% RSLogix 500 project SOL7.RSS, saved by version 8.30.00.16 %
PROJECT "PROJ7"    % processor: Bul.1763 MicroLogix 1100 Series B %

PROGRAM FILES
  LAD 2 "MAIN"  6 rungs
  LAD 3 "IO"  5 rungs
  LAD 4 "CONTROL"  3 rungs
  LAD 5 "CALIBRATE"  8 rungs
  LAD 6 "CYCLE"  2 rungs

DATA FILES
  O0 OUTPUT  4 elements
  I1 INPUT  6 elements
  S2 STATUS  66 elements
  B3 BINARY  1 elements
  T4 TIMER  4 elements
  C5 COUNTER  2 elements
  R6 CONTROL  1 elements
  N7 INTEGER  8 elements
  F8 FLOAT  9 elements

LADDER 2 "MAIN"
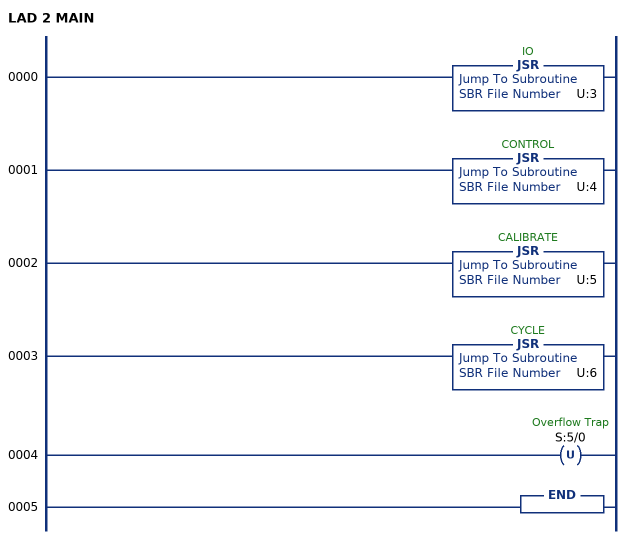
% Rung: 0 %
SOR JSR U:3 EOR
%   U:3  "IO" %
% Rung: 1 %
SOR JSR U:4 EOR
%   U:4  "CONTROL" %
% Rung: 2 %
SOR JSR U:5 EOR
%   U:5  "CALIBRATE" %
% Rung: 3 %
SOR JSR U:6 EOR
%   U:6  "CYCLE" %
% Rung: 4 %
SOR OTU S:5/0 EOR
%   S:5/0  "Overflow Trap" %
% Rung: 5 %
SOR END EOR

LADDER 3 "IO"
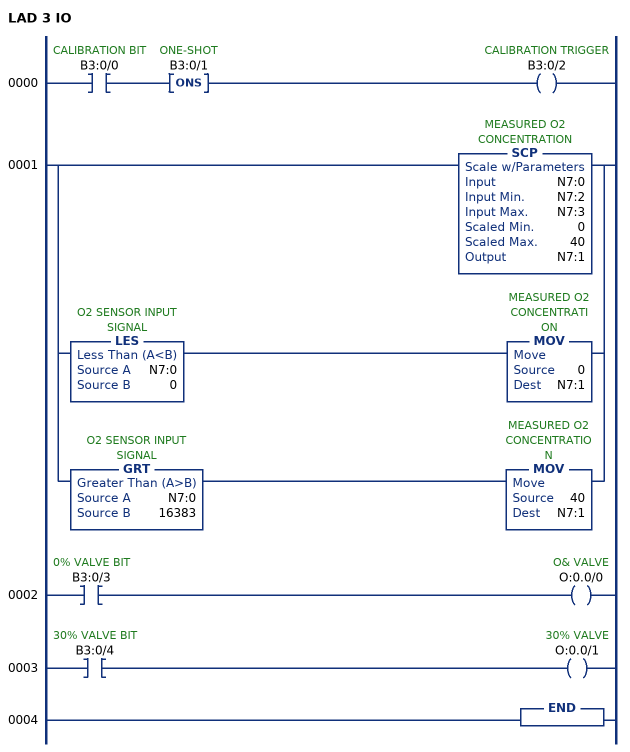
% Rung: 0 %
SOR XIC B3:0/0 ONS B3:0/1 OTE B3:0/2 EOR
%   B3:0/0  "CALIBRATION BIT" %
%   B3:0/1  "ONE-SHOT" %
%   B3:0/2  "CALIBRATION TRIGGER" %
% Rung: 1 %
SOR BST SCP N7:0 N7:2 N7:3 0 40 N7:1 NXB LES N7:0 0 MOV 0 N7:1 NXB GRT N7:0 16383 MOV 40 N7:1 BND EOR
%   N7:0  "O2 SENSOR INPUT SIGNAL" %
%   N7:2  "O2 INPUT MIN" %
%   N7:3  "O2 INPUT MAX" %
%   N7:1  "MEASURED O2 CONCENTRATION" %
% Rung: 2 %
SOR XIC B3:0/3 OTE O:0.0/0 EOR
%   B3:0/3  "0% VALVE BIT" %
%   O:0.0/0  "O& VALVE" %
% Rung: 3 %
SOR XIC B3:0/4 OTE O:0.0/1 EOR
%   B3:0/4  "30% VALVE BIT" %
%   O:0.0/1  "30% VALVE" %
% Rung: 4 %
SOR END EOR

LADDER 4 "CONTROL"
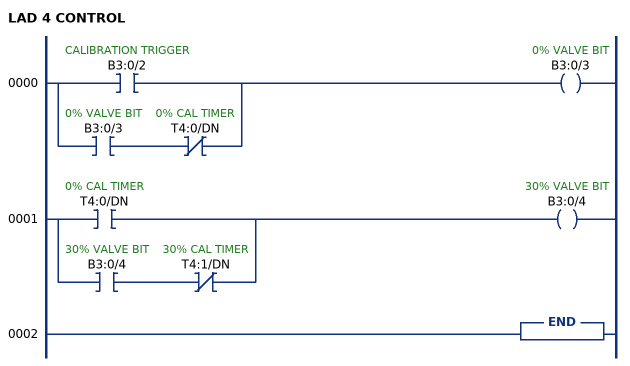
% Rung: 0 %
SOR BST XIC B3:0/2 NXB XIC B3:0/3 XIO T4:0/DN BND OTE B3:0/3 EOR
%   B3:0/2  "CALIBRATION TRIGGER" %
%   B3:0/3  "0% VALVE BIT" %
%   T4:0  "0% CAL TIMER" %
% Rung: 1 %
SOR BST XIC T4:0/DN NXB XIC B3:0/4 XIO T4:1/DN BND OTE B3:0/4 EOR
%   T4:0  "0% CAL TIMER" %
%   B3:0/4  "30% VALVE BIT" %
%   T4:1  "30% CAL TIMER" %
% Rung: 2 %
SOR END EOR

LADDER 5 "CALIBRATE"
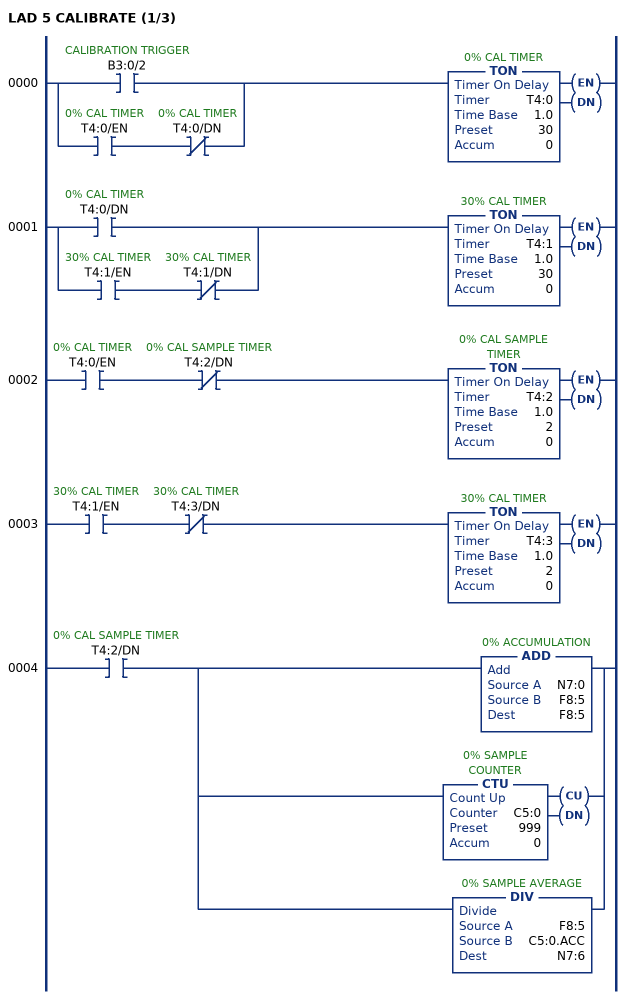
% Rung: 0 %
SOR BST XIC B3:0/2 NXB XIC T4:0/EN XIO T4:0/DN BND TON T4:0 1.0 30 0 EOR
%   B3:0/2  "CALIBRATION TRIGGER" %
%   T4:0  "0% CAL TIMER" %
% Rung: 1 %
SOR BST XIC T4:0/DN NXB XIC T4:1/EN XIO T4:1/DN BND TON T4:1 1.0 30 0 EOR
%   T4:0  "0% CAL TIMER" %
%   T4:1  "30% CAL TIMER" %
% Rung: 2 %
SOR XIC T4:0/EN XIO T4:2/DN TON T4:2 1.0 2 0 EOR
%   T4:0  "0% CAL TIMER" %
%   T4:2  "0% CAL SAMPLE TIMER" %
% Rung: 3 %
SOR XIC T4:1/EN XIO T4:3/DN TON T4:3 1.0 2 0 EOR
%   T4:1  "30% CAL TIMER" %
%   T4:3  "30% CAL TIMER" %
% Rung: 4 %
SOR XIC T4:2/DN BST ADD N7:0 F8:5 F8:5 NXB CTU C5:0 999 0 NXB DIV F8:5 C5:0.ACC N7:6 BND EOR
%   T4:2  "0% CAL SAMPLE TIMER" %
%   N7:0  "O2 SENSOR INPUT SIGNAL" %
%   F8:5  "0% ACCUMULATION" %
%   C5:0  "0% SAMPLE COUNTER" %
%   N7:6  "0% SAMPLE AVERAGE" %

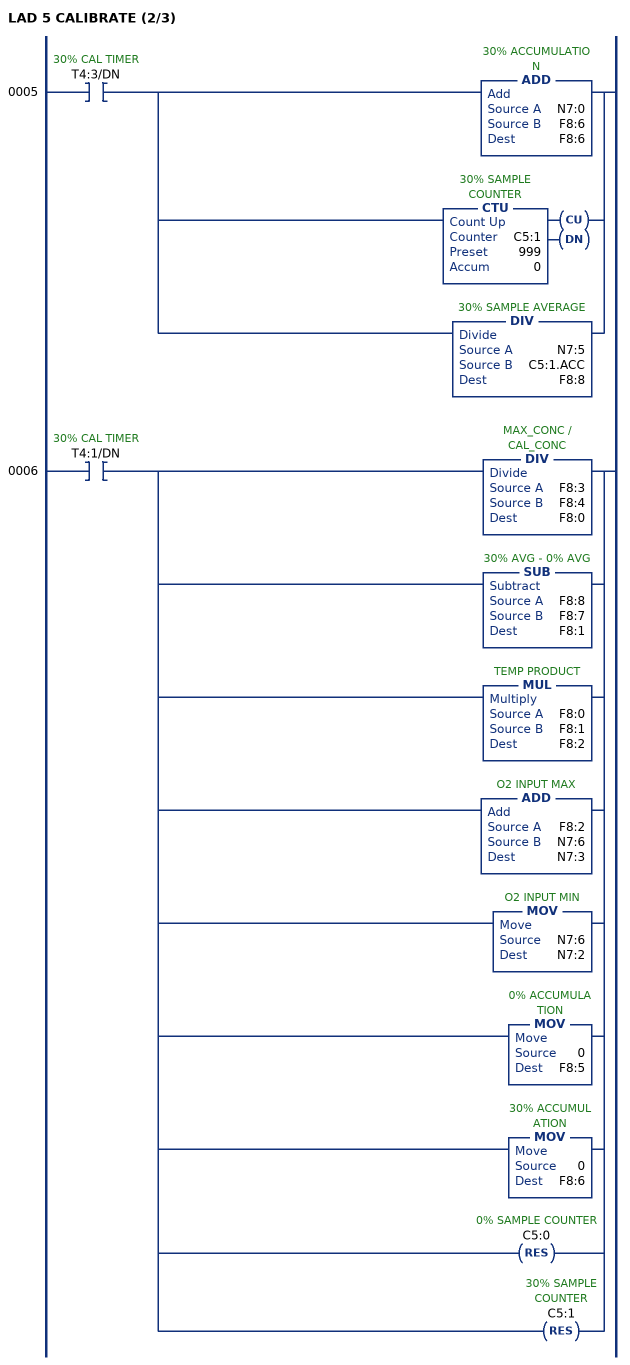
% Rung: 5 %
SOR XIC T4:3/DN BST ADD N7:0 F8:6 F8:6 NXB CTU C5:1 999 0 NXB DIV N7:5 C5:1.ACC F8:8 BND EOR
%   T4:3  "30% CAL TIMER" %
%   N7:0  "O2 SENSOR INPUT SIGNAL" %
%   F8:6  "30% ACCUMULATION" %
%   C5:1  "30% SAMPLE COUNTER" %
%   N7:5  "30% ACCUMULATION" %
%   F8:8  "30% SAMPLE AVERAGE" %
% Rung: 6 %
SOR XIC T4:1/DN BST DIV F8:3 F8:4 F8:0 NXB SUB F8:8 F8:7 F8:1 NXB MUL F8:0 F8:1 F8:2 NXB ADD F8:2 N7:6 N7:3 NXB MOV N7:6 N7:2 NXB MOV 0 F8:5 NXB MOV 0 F8:6 NXB RES C5:0 NXB RES C5:1 BND EOR
%   T4:1  "30% CAL TIMER" %
%   F8:3  "MAX CONCENTRATION" %
%   F8:4  "CAL CONCENTRATION" %
%   F8:0  "MAX_CONC / CAL_CONC" %
%   F8:8  "30% SAMPLE AVERAGE" %
%   F8:7  "30% SAMPLE AVERAGE" %
%   F8:1  "30% AVG - 0% AVG" %
%   F8:2  "TEMP PRODUCT" %
%   N7:6  "0% SAMPLE AVERAGE" %
%   N7:3  "O2 INPUT MAX" %
%   N7:2  "O2 INPUT MIN" %
%   F8:5  "0% ACCUMULATION" %
%   F8:6  "30% ACCUMULATION" %
%   C5:0  "0% SAMPLE COUNTER" %
%   C5:1  "30% SAMPLE COUNTER" %

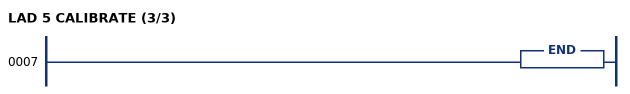
% Rung: 7 %
SOR END EOR

LADDER 6 "CYCLE"
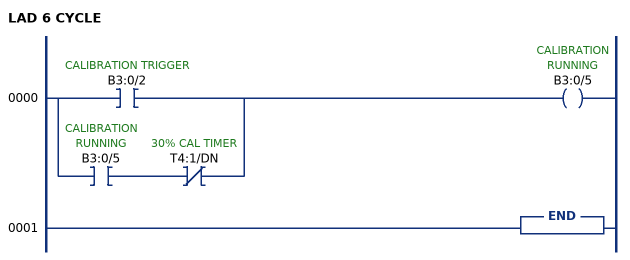
% Rung: 0 %
SOR BST XIC B3:0/2 NXB XIC B3:0/5 XIO T4:1/DN BND OTE B3:0/5 EOR
%   B3:0/2  "CALIBRATION TRIGGER" %
%   B3:0/5  "CALIBRATION RUNNING" %
%   T4:1  "30% CAL TIMER" %
% Rung: 1 %
SOR END EOR

OTHER DOCUMENTED ADDRESSES
  B3:0/6  "CALIBRATION INTERRUPT"
  N7:4  "0% ACCUMULATION"
  N7:7  "30% SAMPLE AVERAGE"
  U:2  "IO"

DATA TABLE (non-zero values as saved)
DATA T4
% .PRE .ACC %
% T4:0 % 30 0
% T4:1 % 30 0
% T4:2 % 2 0
% T4:3 % 2 0
DATA C5
% .PRE .ACC %
% C5:0 % 999 0
% C5:1 % 999 0
DATA F8
% F8:0 % 0 0 0 40 30
